FUNCTION_BLOCK MoveAbsTask IMPLEMENTS I_Task, I_Cyclic, I_Object, I_Abortable
VAR_INPUT
END_VAR
VAR_OUTPUT
END_VAR
VAR
	moveAbs : ARRAY[0..1] OF MoveAbs;
	iMoveAbs : I_MoveAbs := MoveAbs[0];
	moveIndex : INT;
	_Axis : REFERENCE TO AXIS_REF;
END_VAR

{analysis -2}

METHOD Abort : HRESULT
iMoveAbs.Execute := FALSE;
iMoveAbs.Position := 0;
iMoveAbs.Velocity := 0;
END_METHOD

PROPERTY PUBLIC Acceleration : mc_lreal
GET
Acceleration := moveAbs[0].Acceleration;
END_GET
SET
MoveAbs[0].Acceleration := Acceleration;
MoveAbs[1].Acceleration := Acceleration;
END_SET
END_PROPERTY

PROPERTY AxisRef : reference to Axis_Ref
GET // PUBLIC
AxisRef REF= _Axis;
END_GET
SET
_Axis REF= AxisRef;
END_SET
END_PROPERTY

PROPERTY BufferMode : MC_BufferMode
GET
BufferMode := MoveAbs[0].BufferMode;
END_GET
SET
MoveAbs[0].BufferMode := BufferMode;
MoveAbs[1].BufferMode := BufferMode;
END_SET
END_PROPERTY

PROPERTY Busy : BOOL
GET
Busy := iMoveAbs.Busy;
END_GET
END_PROPERTY

METHOD Cycle : HRESULT
VAR_INPUT
END_VAR
moveAbs[0](Axis := _Axis);
moveAbs[1](Axis := _Axis);

iMoveAbs.Execute := FALSE;
END_METHOD

PROPERTY PUBLIC Deceleration : mc_lreal
GET
Deceleration := MoveAbs[0].Deceleration;
END_GET
SET
MoveAbs[0].Deceleration := Deceleration;
MoveAbs[1].Deceleration := Deceleration;
END_SET
END_PROPERTY

PROPERTY Done : BOOL
GET
Done := iMoveAbs.Done;
END_GET
END_PROPERTY

PROPERTY Error : BOOL
GET
Error := iMoveAbs.Error;
END_GET
END_PROPERTY

PROPERTY PUBLIC Jerk : mc_lreal
GET
Jerk := MoveAbs[0].Jerk;
END_GET
SET
MoveAbs[0].Jerk := Jerk;
MoveAbs[1].Jerk := Jerk;
END_SET
END_PROPERTY

METHOD MoveTo : HRESULT
VAR_INPUT
	Position : MC_LREAL;
	Velocity : MC_LREAL;
END_VAR
IF Velocity <= 0.0 THEN
	MoveTo := -1;
	RETURN;
END_IF
Abort();
IF moveIndex = 0 THEN
	moveIndex := 1;
ELSE
	moveIndex := 0;
END_IF
iMoveAbs := moveAbs[moveIndex];
iMoveAbs.Execute := TRUE;
iMoveAbs.Position := Position;
iMoveAbs.Velocity := Velocity;
END_METHOD

METHOD RegisterWithParent
VAR_INPUT
	Parent	: I_HostObjects;
END_VAR
Parent.RegisterAbortable(THIS^);
Parent.RegisterCyclic(THIS^);
Parent.RegisterTask(THIS^);
END_METHOD

END_FUNCTION_BLOCK

(* stored: Version 1.1.0.1
   POU MoveAbsTask: Id {f623c473-a640-4427-8dfd-9222a646d8bd}, SpecialFunc None
   Method Abort: Id {8b24167d-3de8-4038-a0ad-20669890299c}
   Property Acceleration: Id {341f2499-163a-45c5-b240-f5c5cb02dff1}
   Get Get: Id {94f7a0b4-ef99-47e5-9f88-308be92cdbc4}
   Set Set: Id {dbd4bb19-bac7-45a6-9010-56d55b847137}
   Property AxisRef: Id {e141f12b-9dd5-4395-b585-4b5173740d32}
   Get Get: Id {1d6daee9-b5ff-4fb4-b2be-74788b77406f}
   Set Set: Id {9274845b-c3a7-44be-aeb2-ebbc6ead7d6a}
   Property BufferMode: Id {a7c0ed0c-36d3-453f-9975-ca4c3a7e9ba5}
   Get Get: Id {c282e09e-a818-4264-8f8d-0683a728c165}
   Set Set: Id {3591ccd7-2624-4277-b08d-05bb698ae34e}
   Property Busy: Id {1af2a4f9-8f2c-47f1-8f84-24d1cc3c56cc}
   Get Get: Id {d60afff3-b571-480e-8382-7cb6dec1c3d4}
   Method Cycle: Id {968b2426-4712-4973-a44f-8ea7571f0394}
   Property Deceleration: Id {15394e2a-7137-47ee-a0e9-ae4c783d030d}
   Get Get: Id {b409354e-6bdb-432b-bfed-d7faeda4d824}
   Set Set: Id {acdbbe46-8929-47eb-922e-1d284d954e8a}
   Property Done: Id {2efd6afe-2e1a-4877-9647-5bc5cdd99fbe}
   Get Get: Id {e37ef1fe-c5a1-4ddb-9b9d-cdaa750d2b2b}
   Property Error: Id {13f38694-36f8-4930-ab75-64619c3226f8}
   Get Get: Id {be92f53e-b6d5-425a-a3c4-51d3f85be2d7}
   Property Jerk: Id {c177883f-4564-4af8-a89b-8c0edf420990}
   Get Get: Id {5a0859c3-34f7-4dae-a686-377d861e0c51}
   Set Set: Id {6d085ea2-9832-4224-ada6-3f46c8535aed}
   Method MoveTo: Id {094fc655-ef28-4681-8db4-7d4b15208bc6}
   Method RegisterWithParent: Id {1d7ba18a-ff6f-404d-87d7-05ac14b202f6} *)
